SYSTEM FactIOControlApp
  (* Version 1.0, 2021-06-10, Tuojian *)
  APPLICATION FactIOControlAppApp
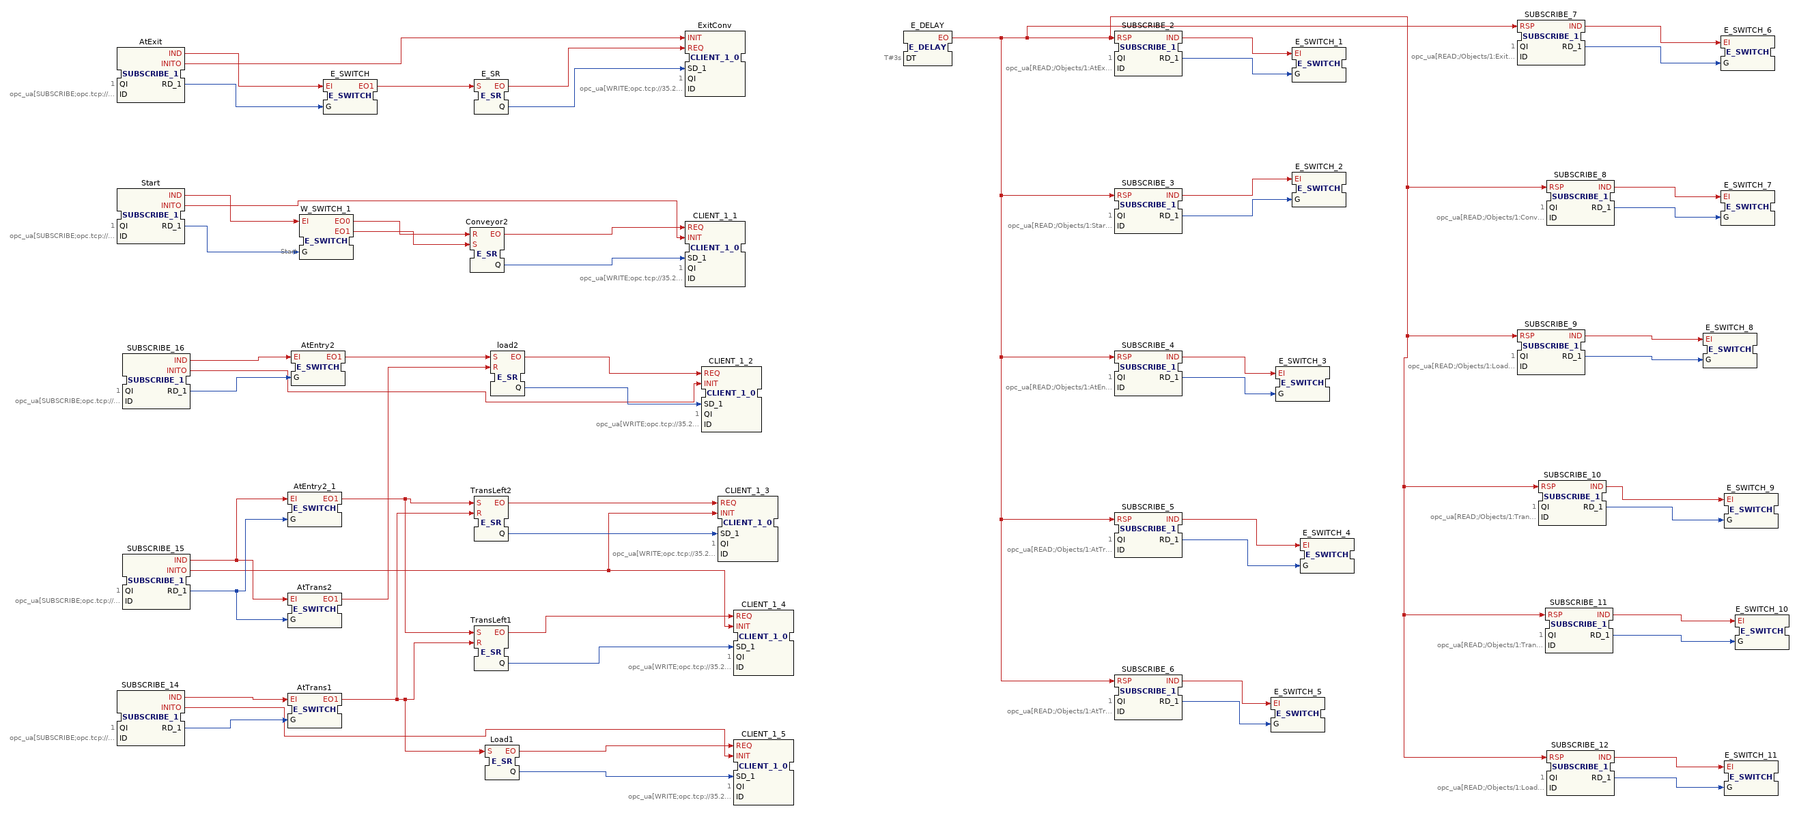
    FBS
      AtExit : SUBSCRIBE_1(QI := 1, ID := opc_ua[SUBSCRIBE;opc.tcp://35.228.36.148:4840#;/Objects/1:AtExit]);
      E_SWITCH : E_SWITCH;
      E_SR : E_SR;
      ExitConv : CLIENT_1_0(QI := 1, ID := opc_ua[WRITE;opc.tcp://35.228.36.148:4840#;/Objects/1:ExitConv]);
      E_DELAY : E_DELAY(DT := T#3s);
      E_SWITCH_1 : E_SWITCH;
      E_SWITCH_2 : E_SWITCH;
      SUBSCRIBE_2 : SUBSCRIBE_1(QI := 1, ID := opc_ua[READ;/Objects/1:AtExit]);
      SUBSCRIBE_3 : SUBSCRIBE_1(QI := 1, ID := opc_ua[READ;/Objects/1:Start]);
      SUBSCRIBE_4 : SUBSCRIBE_1(QI := 1, ID := opc_ua[READ;/Objects/1:AtEntry2]);
      SUBSCRIBE_5 : SUBSCRIBE_1(QI := 1, ID := opc_ua[READ;/Objects/1:AtTrans2]);
      SUBSCRIBE_6 : SUBSCRIBE_1(QI := 1, ID := opc_ua[READ;/Objects/1:AtTrans1]);
      SUBSCRIBE_7 : SUBSCRIBE_1(QI := 1, ID := opc_ua[READ;/Objects/1:ExitConv]);
      SUBSCRIBE_8 : SUBSCRIBE_1(QI := 1, ID := opc_ua[READ;/Objects/1:Conveyor2]);
      SUBSCRIBE_9 : SUBSCRIBE_1(QI := 1, ID := opc_ua[READ;/Objects/1:Load2]);
      SUBSCRIBE_10 : SUBSCRIBE_1(QI := 1, ID := opc_ua[READ;/Objects/1:TransLeft2]);
      SUBSCRIBE_11 : SUBSCRIBE_1(QI := 1, ID := opc_ua[READ;/Objects/1:TransLeft1]);
      SUBSCRIBE_12 : SUBSCRIBE_1(QI := 1, ID := opc_ua[READ;/Objects/1:Load1]);
      E_SWITCH_3 : E_SWITCH;
      E_SWITCH_4 : E_SWITCH;
      E_SWITCH_5 : E_SWITCH;
      E_SWITCH_6 : E_SWITCH;
      E_SWITCH_7 : E_SWITCH;
      E_SWITCH_8 : E_SWITCH;
      E_SWITCH_9 : E_SWITCH;
      E_SWITCH_10 : E_SWITCH;
      E_SWITCH_11 : E_SWITCH;
      TransLeft1 : E_SR;
      Start : SUBSCRIBE_1(QI := 1, ID := opc_ua[SUBSCRIBE;opc.tcp://35.228.36.148:4840#;/Objects/1:Start]);
      Load1 : E_SR;
      AtTrans2 : E_SWITCH;
      TransLeft2 : E_SR;
      SUBSCRIBE_14 : SUBSCRIBE_1(QI := 1, ID := opc_ua[SUBSCRIBE;opc.tcp://35.228.36.148:4840#;/Objects/1:AtTrans1]);
      load2 : E_SR;
      Conveyor2 : E_SR;
      AtTrans1 : E_SWITCH;
      AtEntry2 : E_SWITCH;
      SUBSCRIBE_15 : SUBSCRIBE_1(QI := 1, ID := opc_ua[SUBSCRIBE;opc.tcp://35.228.36.148:4840#;/Objects/1:AtTrans2]);
      AtEntry2_1 : E_SWITCH;
      SUBSCRIBE_16 : SUBSCRIBE_1(QI := 1, ID := opc_ua[SUBSCRIBE;opc.tcp://35.228.36.148:4840#;/Objects/1:AtEntry2]);
      W_SWITCH_1 : E_SWITCH(G := Start);
      CLIENT_1_1 : CLIENT_1_0(QI := 1, ID := opc_ua[WRITE;opc.tcp://35.228.36.148:4840#;/Objects/1:Conveyor2]);
      CLIENT_1_2 : CLIENT_1_0(QI := 1, ID := opc_ua[WRITE;opc.tcp://35.228.36.148:4840#;/Objects/1:Load2]);
      CLIENT_1_3 : CLIENT_1_0(QI := 1, ID := opc_ua[WRITE;opc.tcp://35.228.36.148:4840#;/Objects/1:TransLeft2]);
      CLIENT_1_4 : CLIENT_1_0(QI := 1, ID := opc_ua[WRITE;opc.tcp://35.228.36.148:4840#;/Objects/1:TransLeft1]);
      CLIENT_1_5 : CLIENT_1_0(QI := 1, ID := opc_ua[WRITE;opc.tcp://35.228.36.148:4840#;/Objects/1:Load1]);
    END_FBS
    EVENT_CONNECTIONS
      AtExit.IND TO E_SWITCH.EI;
      AtExit.INITO TO ExitConv.INIT;
      E_SWITCH.EO1 TO E_SR.S;
      E_SR.EO TO ExitConv.REQ;
      E_DELAY.EO TO SUBSCRIBE_2.RSP;
      E_DELAY.EO TO SUBSCRIBE_3.RSP;
      SUBSCRIBE_3.IND TO E_SWITCH_2.EI;
      SUBSCRIBE_2.IND TO E_SWITCH_1.EI;
      E_DELAY.EO TO SUBSCRIBE_4.RSP;
      E_DELAY.EO TO SUBSCRIBE_5.RSP;
      E_DELAY.EO TO SUBSCRIBE_6.RSP;
      E_DELAY.EO TO SUBSCRIBE_7.RSP;
      E_DELAY.EO TO SUBSCRIBE_8.RSP;
      E_DELAY.EO TO SUBSCRIBE_9.RSP;
      E_DELAY.EO TO SUBSCRIBE_10.RSP;
      E_DELAY.EO TO SUBSCRIBE_11.RSP;
      E_DELAY.EO TO SUBSCRIBE_12.RSP;
      SUBSCRIBE_4.IND TO E_SWITCH_3.EI;
      SUBSCRIBE_5.IND TO E_SWITCH_4.EI;
      SUBSCRIBE_6.IND TO E_SWITCH_5.EI;
      SUBSCRIBE_7.IND TO E_SWITCH_6.EI;
      SUBSCRIBE_8.IND TO E_SWITCH_7.EI;
      SUBSCRIBE_9.IND TO E_SWITCH_8.EI;
      SUBSCRIBE_10.IND TO E_SWITCH_9.EI;
      SUBSCRIBE_11.IND TO E_SWITCH_10.EI;
      SUBSCRIBE_12.IND TO E_SWITCH_11.EI;
      AtEntry2_1.EO1 TO TransLeft1.S;
      AtEntry2_1.EO1 TO TransLeft2.S;
      AtEntry2.EO1 TO load2.S;
      W_SWITCH_1.EO0 TO Conveyor2.R;
      AtTrans2.EO1 TO load2.R;
      SUBSCRIBE_15.IND TO AtEntry2_1.EI;
      W_SWITCH_1.EO1 TO Conveyor2.S;
      Start.IND TO W_SWITCH_1.EI;
      AtTrans1.EO1 TO TransLeft2.R;
      AtTrans1.EO1 TO TransLeft1.R;
      SUBSCRIBE_16.IND TO AtEntry2.EI;
      AtTrans1.EO1 TO Load1.S;
      SUBSCRIBE_15.IND TO AtTrans2.EI;
      SUBSCRIBE_14.IND TO AtTrans1.EI;
      Conveyor2.EO TO CLIENT_1_1.REQ;
      load2.EO TO CLIENT_1_2.REQ;
      TransLeft2.EO TO CLIENT_1_3.REQ;
      TransLeft1.EO TO CLIENT_1_4.REQ;
      Load1.EO TO CLIENT_1_5.REQ;
      Start.INITO TO CLIENT_1_1.INIT;
      SUBSCRIBE_16.INITO TO CLIENT_1_2.INIT;
      SUBSCRIBE_15.INITO TO CLIENT_1_3.INIT;
      SUBSCRIBE_15.INITO TO CLIENT_1_4.INIT;
      SUBSCRIBE_14.INITO TO CLIENT_1_5.INIT;
    END_CONNECTIONS
    DATA_CONNECTIONS
      AtExit.RD_1 TO E_SWITCH.G;
      E_SR.Q TO ExitConv.SD_1;
      SUBSCRIBE_2.RD_1 TO E_SWITCH_1.G;
      SUBSCRIBE_3.RD_1 TO E_SWITCH_2.G;
      SUBSCRIBE_4.RD_1 TO E_SWITCH_3.G;
      SUBSCRIBE_5.RD_1 TO E_SWITCH_4.G;
      SUBSCRIBE_6.RD_1 TO E_SWITCH_5.G;
      SUBSCRIBE_7.RD_1 TO E_SWITCH_6.G;
      SUBSCRIBE_8.RD_1 TO E_SWITCH_7.G;
      SUBSCRIBE_9.RD_1 TO E_SWITCH_8.G;
      SUBSCRIBE_10.RD_1 TO E_SWITCH_9.G;
      SUBSCRIBE_11.RD_1 TO E_SWITCH_10.G;
      SUBSCRIBE_12.RD_1 TO E_SWITCH_11.G;
      SUBSCRIBE_15.RD_1 TO AtTrans2.G;
      SUBSCRIBE_15.RD_1 TO AtEntry2_1.G;
      SUBSCRIBE_14.RD_1 TO AtTrans1.G;
      Start.RD_1 TO W_SWITCH_1.G;
      SUBSCRIBE_16.RD_1 TO AtEntry2.G;
      Conveyor2.Q TO CLIENT_1_1.SD_1;
      load2.Q TO CLIENT_1_2.SD_1;
      TransLeft2.Q TO CLIENT_1_3.SD_1;
      TransLeft1.Q TO CLIENT_1_4.SD_1;
      Load1.Q TO CLIENT_1_5.SD_1;
    END_CONNECTIONS
  END_APPLICATION
  DEVICE FORTE_PC : FORTE_PC(MGR_ID := "35.228.36.148:61499")
    {SET_ATTRIBUTE(Profile, HOLOBLOC)} (* device profile *)
    RESOURCE EMB_RES : EMB_RES
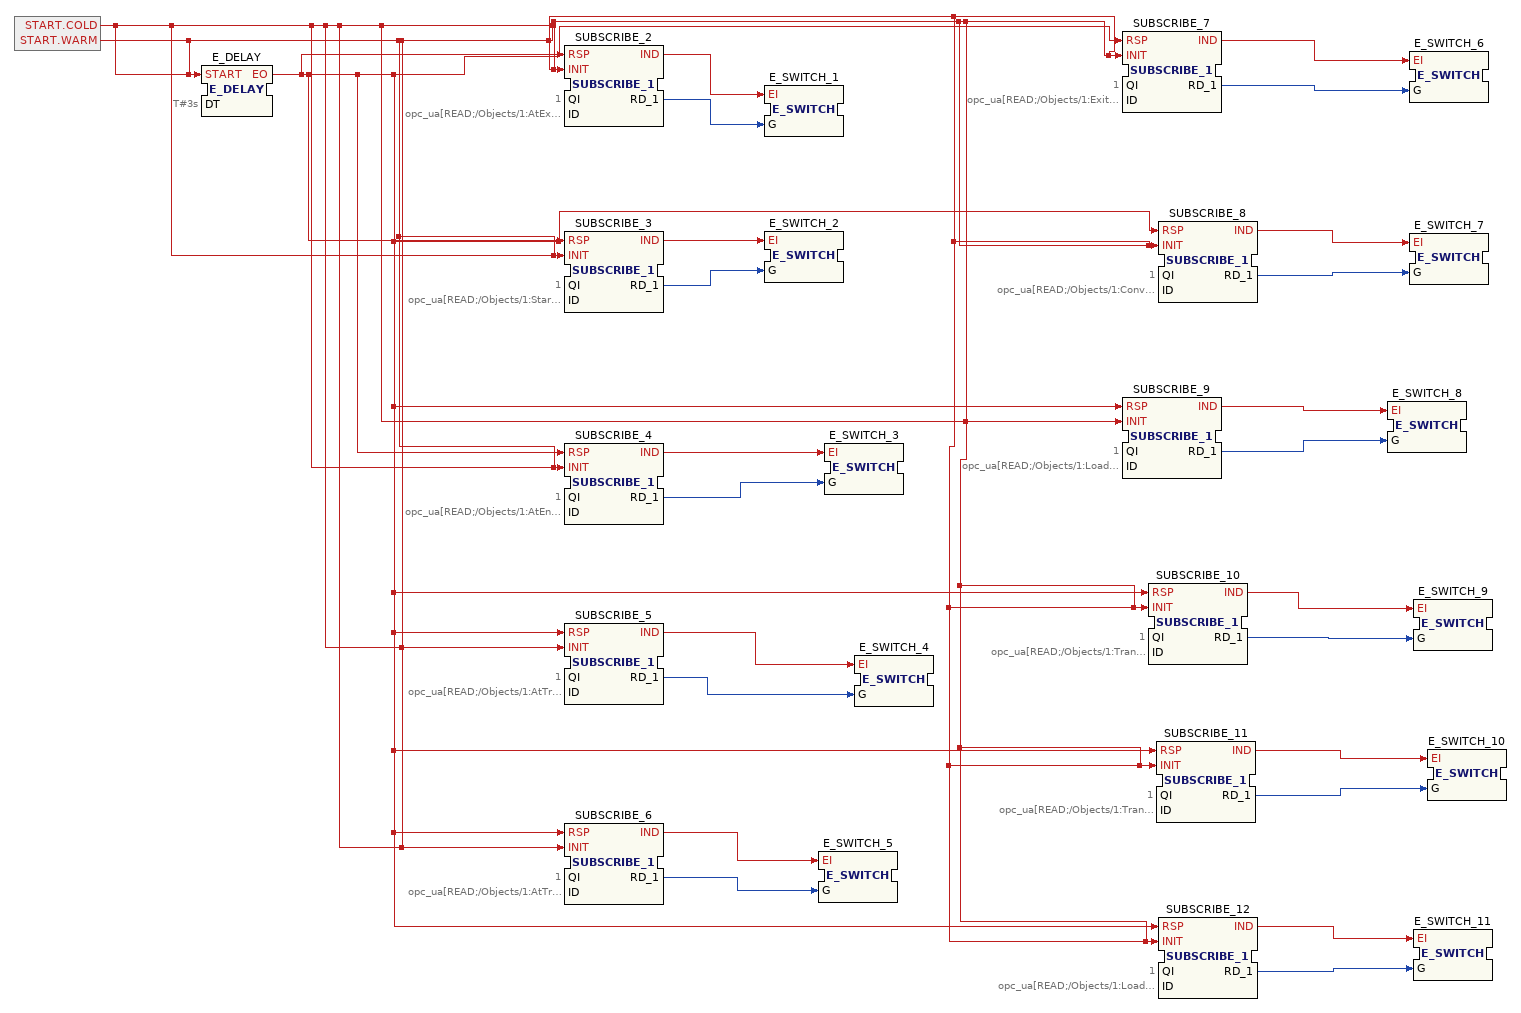
      FBS
        E_DELAY : E_DELAY(DT := T#3s);
        E_SWITCH_1 : E_SWITCH;
        E_SWITCH_2 : E_SWITCH;
        SUBSCRIBE_2 : SUBSCRIBE_1(QI := 1, ID := opc_ua[READ;/Objects/1:AtExit]);
        SUBSCRIBE_3 : SUBSCRIBE_1(QI := 1, ID := opc_ua[READ;/Objects/1:Start]);
        E_SWITCH_7 : E_SWITCH;
        E_SWITCH_6 : E_SWITCH;
        SUBSCRIBE_4 : SUBSCRIBE_1(QI := 1, ID := opc_ua[READ;/Objects/1:AtEntry2]);
        SUBSCRIBE_12 : SUBSCRIBE_1(QI := 1, ID := opc_ua[READ;/Objects/1:Load1]);
        E_SWITCH_3 : E_SWITCH;
        SUBSCRIBE_8 : SUBSCRIBE_1(QI := 1, ID := opc_ua[READ;/Objects/1:Conveyor2]);
        E_SWITCH_11 : E_SWITCH;
        SUBSCRIBE_6 : SUBSCRIBE_1(QI := 1, ID := opc_ua[READ;/Objects/1:AtTrans1]);
        E_SWITCH_5 : E_SWITCH;
        E_SWITCH_4 : E_SWITCH;
        SUBSCRIBE_7 : SUBSCRIBE_1(QI := 1, ID := opc_ua[READ;/Objects/1:ExitConv]);
        SUBSCRIBE_9 : SUBSCRIBE_1(QI := 1, ID := opc_ua[READ;/Objects/1:Load2]);
        SUBSCRIBE_10 : SUBSCRIBE_1(QI := 1, ID := opc_ua[READ;/Objects/1:TransLeft2]);
        E_SWITCH_10 : E_SWITCH;
        SUBSCRIBE_5 : SUBSCRIBE_1(QI := 1, ID := opc_ua[READ;/Objects/1:AtTrans2]);
        SUBSCRIBE_11 : SUBSCRIBE_1(QI := 1, ID := opc_ua[READ;/Objects/1:TransLeft1]);
        E_SWITCH_9 : E_SWITCH;
        E_SWITCH_8 : E_SWITCH;
      END_FBS
      EVENT_CONNECTIONS
        START.COLD TO E_DELAY.START;
        START.WARM TO E_DELAY.START;
        E_DELAY.EO TO SUBSCRIBE_2.RSP;
        E_DELAY.EO TO SUBSCRIBE_3.RSP;
        SUBSCRIBE_3.IND TO E_SWITCH_2.EI;
        SUBSCRIBE_2.IND TO E_SWITCH_1.EI;
        START.COLD TO SUBSCRIBE_2.INIT;
        START.WARM TO SUBSCRIBE_2.INIT;
        START.COLD TO SUBSCRIBE_3.INIT;
        START.WARM TO SUBSCRIBE_3.INIT;
        E_DELAY.EO TO SUBSCRIBE_4.RSP;
        E_DELAY.EO TO SUBSCRIBE_12.RSP;
        SUBSCRIBE_4.IND TO E_SWITCH_3.EI;
        E_DELAY.EO TO SUBSCRIBE_8.RSP;
        SUBSCRIBE_8.IND TO E_SWITCH_7.EI;
        SUBSCRIBE_12.IND TO E_SWITCH_11.EI;
        E_DELAY.EO TO SUBSCRIBE_6.RSP;
        SUBSCRIBE_6.IND TO E_SWITCH_5.EI;
        E_DELAY.EO TO SUBSCRIBE_7.RSP;
        SUBSCRIBE_7.IND TO E_SWITCH_6.EI;
        E_DELAY.EO TO SUBSCRIBE_9.RSP;
        E_DELAY.EO TO SUBSCRIBE_10.RSP;
        E_DELAY.EO TO SUBSCRIBE_5.RSP;
        SUBSCRIBE_5.IND TO E_SWITCH_4.EI;
        E_DELAY.EO TO SUBSCRIBE_11.RSP;
        SUBSCRIBE_11.IND TO E_SWITCH_10.EI;
        SUBSCRIBE_10.IND TO E_SWITCH_9.EI;
        SUBSCRIBE_9.IND TO E_SWITCH_8.EI;
        START.COLD TO SUBSCRIBE_4.INIT;
        START.WARM TO SUBSCRIBE_4.INIT;
        START.COLD TO SUBSCRIBE_5.INIT;
        START.WARM TO SUBSCRIBE_5.INIT;
        START.COLD TO SUBSCRIBE_6.INIT;
        START.WARM TO SUBSCRIBE_6.INIT;
        START.COLD TO SUBSCRIBE_7.INIT;
        START.WARM TO SUBSCRIBE_7.INIT;
        START.COLD TO SUBSCRIBE_8.INIT;
        START.WARM TO SUBSCRIBE_8.INIT;
        START.COLD TO SUBSCRIBE_9.INIT;
        START.WARM TO SUBSCRIBE_9.INIT;
        START.COLD TO SUBSCRIBE_10.INIT;
        START.WARM TO SUBSCRIBE_10.INIT;
        START.COLD TO SUBSCRIBE_11.INIT;
        START.WARM TO SUBSCRIBE_11.INIT;
        START.COLD TO SUBSCRIBE_12.INIT;
        START.WARM TO SUBSCRIBE_12.INIT;
      END_CONNECTIONS
      DATA_CONNECTIONS
        SUBSCRIBE_2.RD_1 TO E_SWITCH_1.G;
        SUBSCRIBE_3.RD_1 TO E_SWITCH_2.G;
        SUBSCRIBE_4.RD_1 TO E_SWITCH_3.G;
        SUBSCRIBE_8.RD_1 TO E_SWITCH_7.G;
        SUBSCRIBE_12.RD_1 TO E_SWITCH_11.G;
        SUBSCRIBE_6.RD_1 TO E_SWITCH_5.G;
        SUBSCRIBE_7.RD_1 TO E_SWITCH_6.G;
        SUBSCRIBE_5.RD_1 TO E_SWITCH_4.G;
        SUBSCRIBE_11.RD_1 TO E_SWITCH_10.G;
        SUBSCRIBE_10.RD_1 TO E_SWITCH_9.G;
        SUBSCRIBE_9.RD_1 TO E_SWITCH_8.G;
      END_CONNECTIONS
    END_RESOURCE
  END_DEVICE
  DEVICE FORTE_PC_1 : FORTE_PC(MGR_ID := "35.228.36.148:61500")
    {SET_ATTRIBUTE(Profile, HOLOBLOC)} (* device profile *)
    RESOURCE EMB_RES : EMB_RES
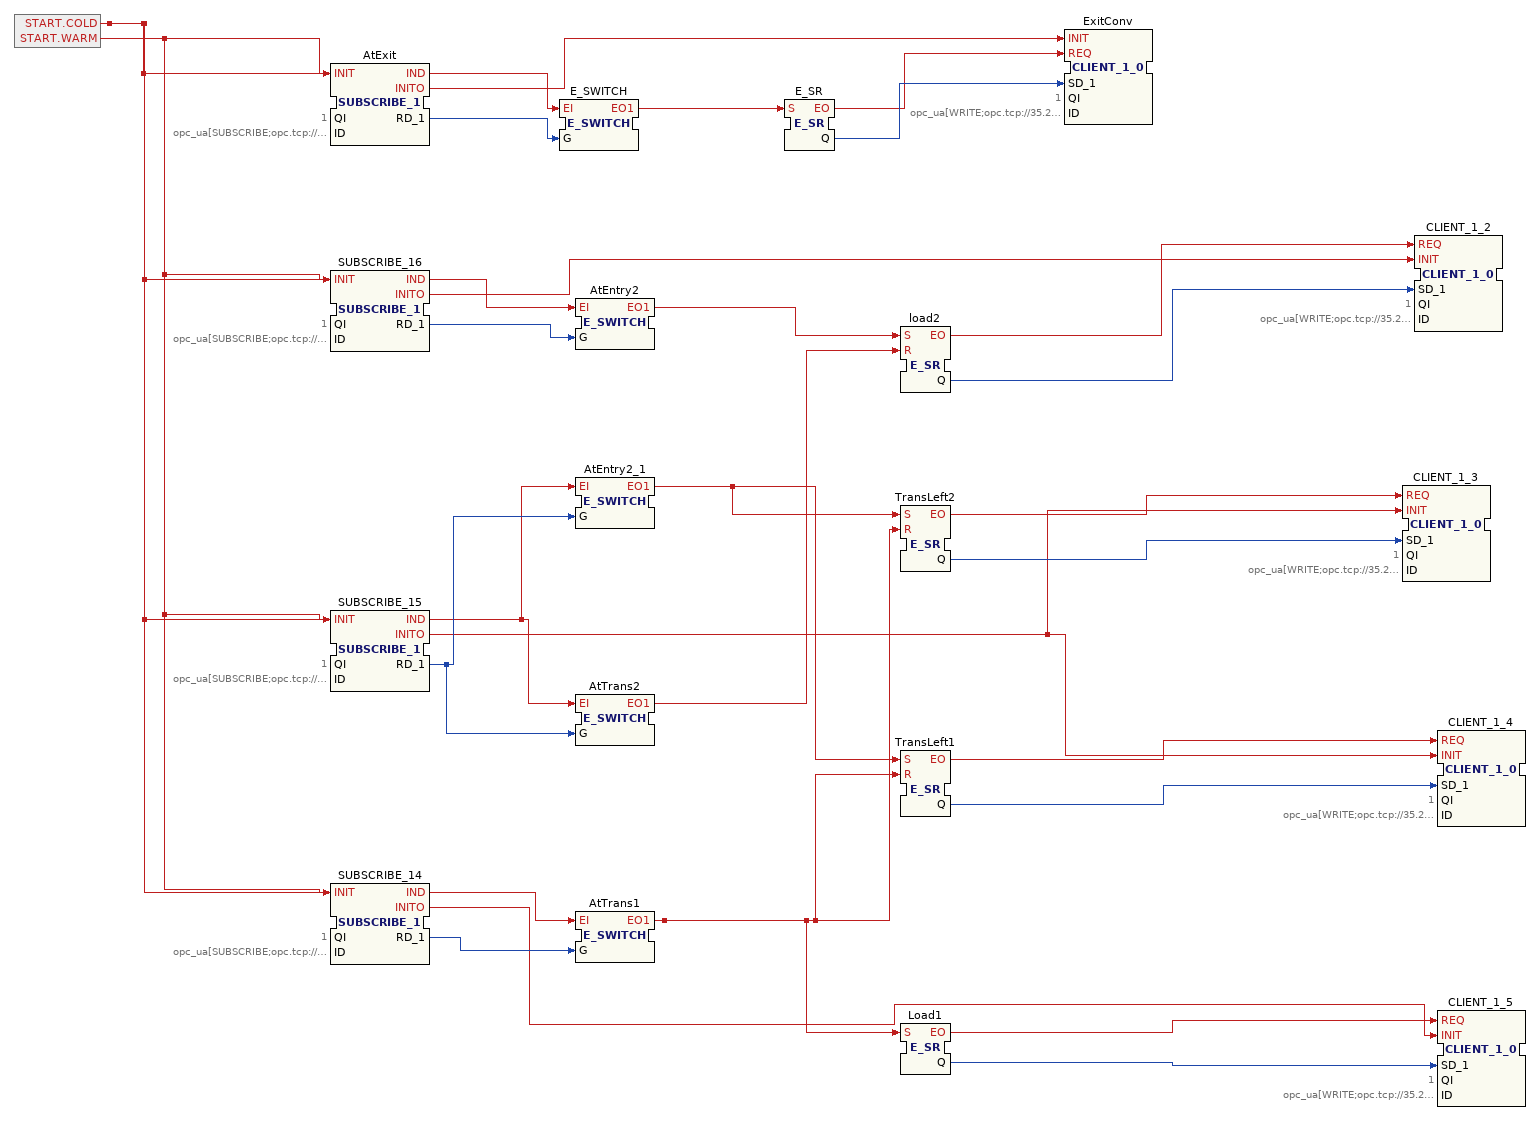
      FBS
        E_SR : E_SR;
        AtExit : SUBSCRIBE_1(QI := 1, ID := opc_ua[SUBSCRIBE;opc.tcp://35.228.36.148:4840#;/Objects/1:AtExit]);
        E_SWITCH : E_SWITCH;
        ExitConv : CLIENT_1_0(QI := 1, ID := opc_ua[WRITE;opc.tcp://35.228.36.148:4840#;/Objects/1:ExitConv]);
        SUBSCRIBE_16 : SUBSCRIBE_1(QI := 1, ID := opc_ua[SUBSCRIBE;opc.tcp://35.228.36.148:4840#;/Objects/1:AtEntry2]);
        AtEntry2 : E_SWITCH;
        CLIENT_1_5 : CLIENT_1_0(QI := 1, ID := opc_ua[WRITE;opc.tcp://35.228.36.148:4840#;/Objects/1:Load1]);
        TransLeft1 : E_SR;
        Load1 : E_SR;
        AtEntry2_1 : E_SWITCH;
        CLIENT_1_2 : CLIENT_1_0(QI := 1, ID := opc_ua[WRITE;opc.tcp://35.228.36.148:4840#;/Objects/1:Load2]);
        TransLeft2 : E_SR;
        AtTrans2 : E_SWITCH;
        SUBSCRIBE_14 : SUBSCRIBE_1(QI := 1, ID := opc_ua[SUBSCRIBE;opc.tcp://35.228.36.148:4840#;/Objects/1:AtTrans1]);
        CLIENT_1_4 : CLIENT_1_0(QI := 1, ID := opc_ua[WRITE;opc.tcp://35.228.36.148:4840#;/Objects/1:TransLeft1]);
        SUBSCRIBE_15 : SUBSCRIBE_1(QI := 1, ID := opc_ua[SUBSCRIBE;opc.tcp://35.228.36.148:4840#;/Objects/1:AtTrans2]);
        AtTrans1 : E_SWITCH;
        CLIENT_1_3 : CLIENT_1_0(QI := 1, ID := opc_ua[WRITE;opc.tcp://35.228.36.148:4840#;/Objects/1:TransLeft2]);
        load2 : E_SR;
      END_FBS
      EVENT_CONNECTIONS
        AtExit.IND TO E_SWITCH.EI;
        E_SWITCH.EO1 TO E_SR.S;
        AtExit.INITO TO ExitConv.INIT;
        E_SR.EO TO ExitConv.REQ;
        START.COLD TO AtExit.INIT;
        START.WARM TO AtExit.INIT;
        SUBSCRIBE_16.IND TO AtEntry2.EI;
        Load1.EO TO CLIENT_1_5.REQ;
        AtEntry2_1.EO1 TO TransLeft1.S;
        AtEntry2_1.EO1 TO TransLeft2.S;
        TransLeft1.EO TO CLIENT_1_4.REQ;
        SUBSCRIBE_15.IND TO AtEntry2_1.EI;
        SUBSCRIBE_15.IND TO AtTrans2.EI;
        SUBSCRIBE_14.IND TO AtTrans1.EI;
        AtTrans1.EO1 TO TransLeft2.R;
        AtTrans1.EO1 TO TransLeft1.R;
        AtTrans1.EO1 TO Load1.S;
        TransLeft2.EO TO CLIENT_1_3.REQ;
        AtEntry2.EO1 TO load2.S;
        AtTrans2.EO1 TO load2.R;
        load2.EO TO CLIENT_1_2.REQ;
        START.COLD TO SUBSCRIBE_16.INIT;
        START.WARM TO SUBSCRIBE_16.INIT;
        START.COLD TO SUBSCRIBE_15.INIT;
        START.WARM TO SUBSCRIBE_15.INIT;
        START.COLD TO SUBSCRIBE_14.INIT;
        START.WARM TO SUBSCRIBE_14.INIT;
        SUBSCRIBE_16.INITO TO CLIENT_1_2.INIT;
        SUBSCRIBE_15.INITO TO CLIENT_1_3.INIT;
        SUBSCRIBE_15.INITO TO CLIENT_1_4.INIT;
        SUBSCRIBE_14.INITO TO CLIENT_1_5.INIT;
      END_CONNECTIONS
      DATA_CONNECTIONS
        AtExit.RD_1 TO E_SWITCH.G;
        E_SR.Q TO ExitConv.SD_1;
        SUBSCRIBE_16.RD_1 TO AtEntry2.G;
        Load1.Q TO CLIENT_1_5.SD_1;
        TransLeft1.Q TO CLIENT_1_4.SD_1;
        SUBSCRIBE_15.RD_1 TO AtTrans2.G;
        SUBSCRIBE_15.RD_1 TO AtEntry2_1.G;
        SUBSCRIBE_14.RD_1 TO AtTrans1.G;
        TransLeft2.Q TO CLIENT_1_3.SD_1;
        load2.Q TO CLIENT_1_2.SD_1;
      END_CONNECTIONS
    END_RESOURCE
  END_DEVICE
  DEVICE FORTE_PC_2 : FORTE_PC(MGR_ID := "35.228.36.148:61501")
    {SET_ATTRIBUTE(Profile, HOLOBLOC)} (* device profile *)
    RESOURCE EMB_RES : EMB_RES
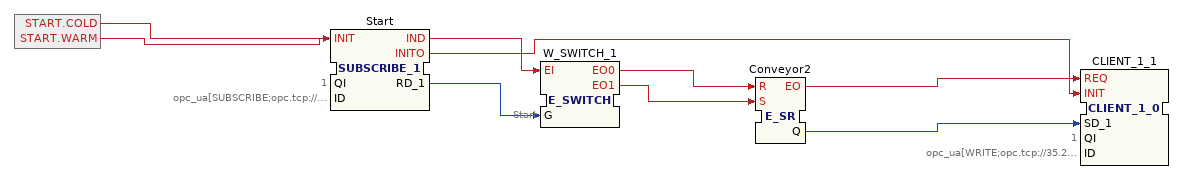
      FBS
        CLIENT_1_1 : CLIENT_1_0(QI := 1, ID := opc_ua[WRITE;opc.tcp://35.228.36.148:4840#;/Objects/1:Conveyor2]);
        Conveyor2 : E_SR;
        W_SWITCH_1 : E_SWITCH(G := Start);
        Start : SUBSCRIBE_1(QI := 1, ID := opc_ua[SUBSCRIBE;opc.tcp://35.228.36.148:4840#;/Objects/1:Start]);
      END_FBS
      EVENT_CONNECTIONS
        Conveyor2.EO TO CLIENT_1_1.REQ;
        W_SWITCH_1.EO0 TO Conveyor2.R;
        W_SWITCH_1.EO1 TO Conveyor2.S;
        Start.IND TO W_SWITCH_1.EI;
        Start.INITO TO CLIENT_1_1.INIT;
        START.COLD TO Start.INIT;
        START.WARM TO Start.INIT;
      END_CONNECTIONS
      DATA_CONNECTIONS
        Conveyor2.Q TO CLIENT_1_1.SD_1;
        Start.RD_1 TO W_SWITCH_1.G;
      END_CONNECTIONS
    END_RESOURCE
  END_DEVICE
  MAPPINGS
    FactIOControlAppApp.E_DELAY ON FORTE_PC.EMB_RES.E_DELAY;
    FactIOControlAppApp.E_SWITCH_1 ON FORTE_PC.EMB_RES.E_SWITCH_1;
    FactIOControlAppApp.E_SR ON FORTE_PC_1.EMB_RES.E_SR;
    FactIOControlAppApp.AtExit ON FORTE_PC_1.EMB_RES.AtExit;
    FactIOControlAppApp.E_SWITCH ON FORTE_PC_1.EMB_RES.E_SWITCH;
    FactIOControlAppApp.ExitConv ON FORTE_PC_1.EMB_RES.ExitConv;
    FactIOControlAppApp.E_SWITCH_2 ON FORTE_PC.EMB_RES.E_SWITCH_2;
    FactIOControlAppApp.SUBSCRIBE_2 ON FORTE_PC.EMB_RES.SUBSCRIBE_2;
    FactIOControlAppApp.SUBSCRIBE_3 ON FORTE_PC.EMB_RES.SUBSCRIBE_3;
    FactIOControlAppApp.E_SWITCH_7 ON FORTE_PC.EMB_RES.E_SWITCH_7;
    FactIOControlAppApp.E_SWITCH_6 ON FORTE_PC.EMB_RES.E_SWITCH_6;
    FactIOControlAppApp.SUBSCRIBE_4 ON FORTE_PC.EMB_RES.SUBSCRIBE_4;
    FactIOControlAppApp.SUBSCRIBE_12 ON FORTE_PC.EMB_RES.SUBSCRIBE_12;
    FactIOControlAppApp.E_SWITCH_3 ON FORTE_PC.EMB_RES.E_SWITCH_3;
    FactIOControlAppApp.SUBSCRIBE_8 ON FORTE_PC.EMB_RES.SUBSCRIBE_8;
    FactIOControlAppApp.E_SWITCH_11 ON FORTE_PC.EMB_RES.E_SWITCH_11;
    FactIOControlAppApp.SUBSCRIBE_6 ON FORTE_PC.EMB_RES.SUBSCRIBE_6;
    FactIOControlAppApp.E_SWITCH_5 ON FORTE_PC.EMB_RES.E_SWITCH_5;
    FactIOControlAppApp.E_SWITCH_4 ON FORTE_PC.EMB_RES.E_SWITCH_4;
    FactIOControlAppApp.SUBSCRIBE_7 ON FORTE_PC.EMB_RES.SUBSCRIBE_7;
    FactIOControlAppApp.SUBSCRIBE_9 ON FORTE_PC.EMB_RES.SUBSCRIBE_9;
    FactIOControlAppApp.SUBSCRIBE_10 ON FORTE_PC.EMB_RES.SUBSCRIBE_10;
    FactIOControlAppApp.E_SWITCH_10 ON FORTE_PC.EMB_RES.E_SWITCH_10;
    FactIOControlAppApp.SUBSCRIBE_5 ON FORTE_PC.EMB_RES.SUBSCRIBE_5;
    FactIOControlAppApp.SUBSCRIBE_11 ON FORTE_PC.EMB_RES.SUBSCRIBE_11;
    FactIOControlAppApp.E_SWITCH_9 ON FORTE_PC.EMB_RES.E_SWITCH_9;
    FactIOControlAppApp.E_SWITCH_8 ON FORTE_PC.EMB_RES.E_SWITCH_8;
    FactIOControlAppApp.CLIENT_1_1 ON FORTE_PC_2.EMB_RES.CLIENT_1_1;
    FactIOControlAppApp.Conveyor2 ON FORTE_PC_2.EMB_RES.Conveyor2;
    FactIOControlAppApp.W_SWITCH_1 ON FORTE_PC_2.EMB_RES.W_SWITCH_1;
    FactIOControlAppApp.Start ON FORTE_PC_2.EMB_RES.Start;
    FactIOControlAppApp.SUBSCRIBE_16 ON FORTE_PC_1.EMB_RES.SUBSCRIBE_16;
    FactIOControlAppApp.AtEntry2 ON FORTE_PC_1.EMB_RES.AtEntry2;
    FactIOControlAppApp.CLIENT_1_5 ON FORTE_PC_1.EMB_RES.CLIENT_1_5;
    FactIOControlAppApp.TransLeft1 ON FORTE_PC_1.EMB_RES.TransLeft1;
    FactIOControlAppApp.Load1 ON FORTE_PC_1.EMB_RES.Load1;
    FactIOControlAppApp.AtEntry2_1 ON FORTE_PC_1.EMB_RES.AtEntry2_1;
    FactIOControlAppApp.CLIENT_1_2 ON FORTE_PC_1.EMB_RES.CLIENT_1_2;
    FactIOControlAppApp.TransLeft2 ON FORTE_PC_1.EMB_RES.TransLeft2;
    FactIOControlAppApp.AtTrans2 ON FORTE_PC_1.EMB_RES.AtTrans2;
    FactIOControlAppApp.SUBSCRIBE_14 ON FORTE_PC_1.EMB_RES.SUBSCRIBE_14;
    FactIOControlAppApp.CLIENT_1_4 ON FORTE_PC_1.EMB_RES.CLIENT_1_4;
    FactIOControlAppApp.SUBSCRIBE_15 ON FORTE_PC_1.EMB_RES.SUBSCRIBE_15;
    FactIOControlAppApp.AtTrans1 ON FORTE_PC_1.EMB_RES.AtTrans1;
    FactIOControlAppApp.CLIENT_1_3 ON FORTE_PC_1.EMB_RES.CLIENT_1_3;
    FactIOControlAppApp.load2 ON FORTE_PC_1.EMB_RES.load2;
  END_MAPPINGS
  SEGMENTS
    Ethernet : Ethernet;
  END_SEGMENTS
  LINKS
    FORTE_PC => Ethernet;
    FORTE_PC_1 => Ethernet;
    FORTE_PC_2 => Ethernet;
  END_LINKS
END_SYSTEM
